{attribute 'qualified_only'}
{attribute 'strict'}
TYPE System_Modus_Enum :
(
	System_Init := 0,
	System_Run
);
END_TYPE

(* stored: Version 1.1.0.1, ProductVersion 3.1.4024.13
   DUT System_Modus_Enum: Id {feb8246f-8f13-4334-9f5f-28a5f9dfb58b} *)
